// TIA Portal V18 export
// export: Created 2025-12-01T12:38:33.4037087Z, ExportSetting None, DisplayName Totally Integrated Automation Portal, DisplayVersion V18 Update 5, DisplayName TIA Portal Openness, DisplayVersion V18 Update 5, DisplayName TIA Portal Teamcenter Gateway, DisplayVersion V18, DisplayName TIA Portal Version Control Interface, DisplayVersion V18, DisplayName STEP 7 Professional, DisplayVersion V18 Update 5, DisplayName STEP 7 Safety, DisplayVersion V18, DisplayName WinCC Professional, DisplayVersion V18 Update 5
FUNCTION "ST10Cyl_interface11-20" : Void   // FC1021, LAD
{ S7_Optimized_Access := 'FALSE' }
// stored: AutoNumber false, SetENOAutomatically false
   VAR_INPUT
      AlwaysON : Bool;
      E_stop : Bool;
   END_VAR
   VAR_TEMP
      tTest : Bool;
   END_VAR
BEGIN

REGION Network 1 (SCL): Cylinder 11-20 IO Interface (SCL)

   //Cylinder11 IO   E-NG-01NGLocationCylinder
   //Input
   "ST10Cylinder".Cy[11].In.WorkPositionSensor := "iE-NG-01NGLocationCylinderInWP";
   "ST10Cylinder".Cy[11].In.HomePositionSensor := "iE-NG-01NGLocationCylinderInHP";
   //Output
   "oE-NG-01NGLocationCylinderToWP" := "ST10Cylinder".Cy[11].Out.GoWorkPosition;
   "oE-NG-01NGLocationCylinderToHP" := "ST10Cylinder".Cy[11].Out.GoHomePosition;

   //Cylinder12 IO  E-NG-02NGLocationCylinder
   //Input
   "ST10Cylinder".Cy[12].In.WorkPositionSensor := "iE-NG-02NGLocationCylinderInWP";
   "ST10Cylinder".Cy[12].In.HomePositionSensor := "iE-NG-02NGLocationCylinderInHP";
   //Output
   "oE-NG-02NGLocationCylinderToWP" := "ST10Cylinder".Cy[12].Out.GoWorkPosition;
   "oE-NG-02NGLocationCylinderToHP" := "ST10Cylinder".Cy[12].Out.GoHomePosition;

   //Cylinder13 IO  F-ROOBT1Gripper1Cylinder
   //Input
   "KukaRobot1_CtrlDB".sPLCtoROB.User.Gripper.DI129_Grip1WP:="ST10Cylinder".Cy[13].In.WorkPositionSensor := "iF-ROOBT1Gripper1CylinderInWP" ;
   "KukaRobot1_CtrlDB".sPLCtoROB.User.Gripper.DI130_Grip1HP := "ST10Cylinder".Cy[13].In.HomePositionSensor := "iF-ROOBT1Gripper1CylinderInHP" ;//"TON".TON[0].Q;

   IF  NOT "Robot_DB".Control.Robot1GripControl THEN
       //Output
       "oF-ROOBT1Gripper1CylinderToWP" := "KukaRobot1_CtrlDB".sROBtoPLC.User.Gripper.DO129_Grip1GoWork;
       "oF-ROOBT1Gripper1CylinderToHP" := "KukaRobot1_CtrlDB".sROBtoPLC.User.Gripper.DO130_Grip1GoHome;
   ELSE
       //Output
       "oF-ROOBT1Gripper1CylinderToWP" := "ST10Cylinder".Cy[13].Out.GoWorkPosition;
       "oF-ROOBT1Gripper1CylinderToHP" := "ST10Cylinder".Cy[13].Out.GoHomePosition;
   END_IF;
   "TON".TON[0](IN:="oF-ROOBT1Gripper1CylinderToHP" AND NOT"iF-ROOBT1Gripper1CylinderInWP",PT:=T#500MS);


   //Cylinder14 IO  F-ROOBT1Gripper2Cylinder
   //Input
   "KukaRobot1_CtrlDB".sPLCtoROB.User.Gripper.DI131_Grip2WP:="ST10Cylinder".Cy[14].In.WorkPositionSensor := "iF-ROOBT1Gripper2CylinderInWP";
   "KukaRobot1_CtrlDB".sPLCtoROB.User.Gripper.DI132_Grip2HP:="ST10Cylinder".Cy[14].In.HomePositionSensor := "iF-ROOBT1Gripper2CylinderInHP";

   IF NOT "Robot_DB".Control.Robot1GripControl THEN
       //Output
       "oF-ROOBT1Gripper2CylinderToWP" :="ST10Cylinder".Cy[14].Inout.AutoGoWork:="KukaRobot1_CtrlDB".sROBtoPLC.User.Gripper.DO131_Grip2GoWork;
       "oF-ROOBT1Gripper2CylinderToHP" :="ST10Cylinder".Cy[14].Inout.AutoGoHome:="KukaRobot1_CtrlDB".sROBtoPLC.User.Gripper.DO132_Grip2GoHome;
   ELSE
       //Output
       "oF-ROOBT1Gripper2CylinderToWP" := "ST10Cylinder".Cy[14].Out.GoWorkPosition;
       "oF-ROOBT1Gripper2CylinderToHP" := "ST10Cylinder".Cy[14].Out.GoHomePosition;
   END_IF;


   //Cylinder15 IO  F-ROOBT2Gripper1Cylinder
   //Input
   "KukaRobot2_CtrlDB".sPLCtoROB.User.Gripper.DI129_Grip1WP:="ST10Cylinder".Cy[15].In.WorkPositionSensor := "iF-ROOBT2Gripper1CylinderInWP";
   "KukaRobot2_CtrlDB".sPLCtoROB.User.Gripper.DI130_Grip1HP := "ST10Cylinder".Cy[15].In.HomePositionSensor :="iF-ROOBT2Gripper1CylinderInHP";

   IF NOT "Robot_DB".Control.Robot2GripControl THEN
       //Output
       "oF-ROOBT2Gripper1CylinderToWP" :="ST10Cylinder".Cy[15].Inout.AutoGoWork:="KukaRobot2_CtrlDB".sROBtoPLC.User.Gripper.DO129_Grip1GoWork;
       "oF-ROOBT2Gripper1CylinderToHP" :="ST10Cylinder".Cy[15].Inout.AutoGoHome:="KukaRobot2_CtrlDB".sROBtoPLC.User.Gripper.DO130_Grip1GoHome;
   ELSE
       //Output
       "oF-ROOBT2Gripper1CylinderToWP" := "ST10Cylinder".Cy[15].Out.GoWorkPosition;
       "oF-ROOBT2Gripper1CylinderToHP" := "ST10Cylinder".Cy[15].Out.GoHomePosition;
   END_IF;



   //Cylinder16 IO  F-ROOBT2Gripper2Cylinder
   //Input
   "KukaRobot2_CtrlDB".sPLCtoROB.User.Gripper.DI131_Grip2WP:="ST10Cylinder".Cy[16].In.WorkPositionSensor := "iF-ROOBT2Gripper2CylinderInWP";
   "KukaRobot2_CtrlDB".sPLCtoROB.User.Gripper.DI132_Grip2HP:="ST10Cylinder".Cy[16].In.HomePositionSensor := "iF-ROOBT2Gripper2CylinderInHP";

   IF NOT "Robot_DB".Control.Robot2GripControl THEN
       //Output
       "oF-ROOBT2Gripper2CylinderToWP" :="ST10Cylinder".Cy[16].Inout.AutoGoWork:= "KukaRobot2_CtrlDB".sROBtoPLC.User.Gripper.DO131_Grip2GoWork;
       "oF-ROOBT2Gripper2CylinderToHP" :="ST10Cylinder".Cy[16].Inout.AutoGoHome:= "KukaRobot2_CtrlDB".sROBtoPLC.User.Gripper.DO132_Grip2GoHome;
   ELSE
       //Output
       "oF-ROOBT2Gripper2CylinderToWP" := "ST10Cylinder".Cy[16].Out.GoWorkPosition;
       "oF-ROOBT2Gripper2CylinderToHP" := "ST10Cylinder".Cy[16].Out.GoHomePosition;
   END_IF;

   //Cylinder17 IO  F-ROOBT3Gripper1Cylinder
   //Input
   "KukaRobot3_CtrlDB".sPLCtoROB.User.Gripper.DI129_Grip1WP:="ST10Cylinder".Cy[17].In.WorkPositionSensor := "iF-ROOBT3Gripper1CylinderInWP";
   "KukaRobot3_CtrlDB".sPLCtoROB.User.Gripper.DI130_Grip1HP:="ST10Cylinder".Cy[17].In.HomePositionSensor := "iF-ROOBT3Gripper1CylinderInHP";

   IF NOT "Robot_DB".Control.Robot3GripControl THEN
       //Output
       "oF-ROOBT3Gripper1CylinderToWP" :="ST10Cylinder".Cy[17].Inout.AutoGoWork:="KukaRobot3_CtrlDB".sROBtoPLC.User.Gripper.DO129_Grip1GoWork;
       "oF-ROOBT3Gripper1CylinderToHP" :="ST10Cylinder".Cy[17].Inout.AutoGoHome:="KukaRobot3_CtrlDB".sROBtoPLC.User.Gripper.DO130_Grip1GoHome;
   ELSE
       //Output
       "oF-ROOBT3Gripper1CylinderToWP" := "ST10Cylinder".Cy[17].Out.GoWorkPosition;
       "oF-ROOBT3Gripper1CylinderToHP" := "ST10Cylinder".Cy[17].Out.GoHomePosition;
   END_IF;


   //Cylinder18 IO  F-ROOBT3Gripper2Cylinder
   //Input
   "KukaRobot3_CtrlDB".sPLCtoROB.User.Gripper.DI131_Grip2WP:="ST10Cylinder".Cy[18].In.WorkPositionSensor := "iF-ROOBT3Gripper2CylinderInWP";
   "KukaRobot3_CtrlDB".sPLCtoROB.User.Gripper.DI132_Grip2HP := "ST10Cylinder".Cy[18].In.HomePositionSensor := "iF-ROOBT3Gripper2CylinderInHP";//"TON".TON[1].Q;

   IF NOT "Robot_DB".Control.Robot3GripControl THEN
       //Output
       "oF-ROOBT3Gripper2CylinderToWP" :="ST10Cylinder".Cy[18].Inout.AutoGoWork:="KukaRobot3_CtrlDB".sROBtoPLC.User.Gripper.DO131_Grip2GoWork;
       "oF-ROOBT3Gripper2CylinderToHP" :="ST10Cylinder".Cy[18].Inout.AutoGoHome:="KukaRobot3_CtrlDB".sROBtoPLC.User.Gripper.DO132_Grip2GoHome;
   ELSE
       //Output
       "oF-ROOBT3Gripper2CylinderToWP" := "ST10Cylinder".Cy[18].Out.GoWorkPosition;
       "oF-ROOBT3Gripper2CylinderToHP" := "ST10Cylinder".Cy[18].Out.GoHomePosition;
   END_IF;

   "TON".TON[1](IN := "oF-ROOBT3Gripper2CylinderToHP" AND NOT "iF-ROOBT3Gripper2CylinderInWP",
                PT := T#500MS);

   (*
   //Cylinder19 IO  D-washer Loading Horizontal
   //Input
   "ST10Cylinder".Cy[19].In.WorkPositionSensor := ("D-washer Loading Cylinder Middle Cylinder InHP" AND "D-washer Loading Horizontal Cylinder InWP")
                                               OR ("D-washer Loading Cylinder Middle Cylinder InWP" AND "D-washer Loading Horizontal Cylinder InWP1");
   "ST10Cylinder".Cy[19].In.HomePositionSensor := "D-washer Loading Horizontal Cylinder InHP";
   //Output
   "D-washer Loading Horizontal Cylinder ToWP" := "ST10Cylinder".Cy[19].Out.GoWorkPosition;
   "D-washer Loading Horizontal Cylinder ToHP" := "ST10Cylinder".Cy[19].Out.GoHomePosition;

   //Cylinder20 IO  D-washer Loading Cylinder Middle
   //Input
   "ST10Cylinder".Cy[20].In.WorkPositionSensor := "D-washer Loading Cylinder Middle Cylinder InWP";
   "ST10Cylinder".Cy[20].In.HomePositionSensor := "D-washer Loading Cylinder Middle Cylinder InHP";
   //Output
   "D-washer Loading Cylinder Middle Cylinder ToWP" := "ST10Cylinder".Cy[20].Out.GoWorkPosition;
   "D-washer Loading Cylinder Middle Cylinder ToHP" := "ST10Cylinder".Cy[20].Out.GoHomePosition;
   *)
END_REGION

REGION Network 2: CY11 interface E-NG-01NGLocationCylinder
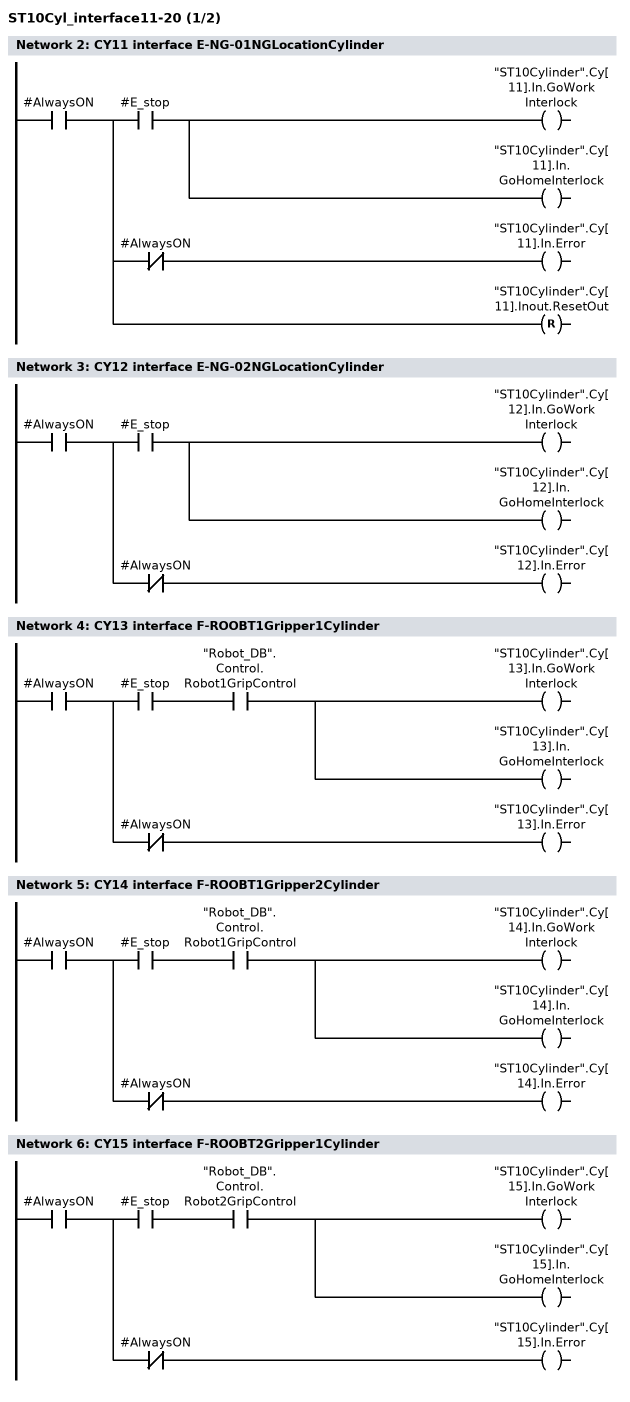
   RUNG wire#powerrail
      Contact( #AlwaysON )
      wire#w1
      Contact( #E_stop )
      wire#w2
      Coil( "ST10Cylinder".Cy[11].In.GoWorkInterlock )
   END_RUNG
   RUNG wire#w2
      Coil( "ST10Cylinder".Cy[11].In.GoHomeInterlock )
   END_RUNG
   RUNG wire#w1
      I_Contact( #AlwaysON )
      Coil( "ST10Cylinder".Cy[11].In.Error )
   END_RUNG
   RUNG wire#w1
      R_Coil( "ST10Cylinder".Cy[11].Inout.ResetOut )
   END_RUNG
   // the same network as SCL:
   "ST10Cylinder".Cy[11].In.GoWorkInterlock := #AlwaysON AND #E_stop;
   "ST10Cylinder".Cy[11].In.GoHomeInterlock := #AlwaysON AND #E_stop;
   "ST10Cylinder".Cy[11].In.Error := #AlwaysON AND NOT #AlwaysON;
   IF #AlwaysON THEN "ST10Cylinder".Cy[11].Inout.ResetOut := FALSE; END_IF;
END_REGION

REGION Network 3: CY12 interface E-NG-02NGLocationCylinder
   RUNG wire#powerrail
      Contact( #AlwaysON )
      wire#w1
      Contact( #E_stop )
      wire#w2
      Coil( "ST10Cylinder".Cy[12].In.GoWorkInterlock )
   END_RUNG
   RUNG wire#w2
      Coil( "ST10Cylinder".Cy[12].In.GoHomeInterlock )
   END_RUNG
   RUNG wire#w1
      I_Contact( #AlwaysON )
      Coil( "ST10Cylinder".Cy[12].In.Error )
   END_RUNG
   // the same network as SCL:
   "ST10Cylinder".Cy[12].In.GoWorkInterlock := #AlwaysON AND #E_stop;
   "ST10Cylinder".Cy[12].In.GoHomeInterlock := #AlwaysON AND #E_stop;
   "ST10Cylinder".Cy[12].In.Error := #AlwaysON AND NOT #AlwaysON;
END_REGION

REGION Network 4: CY13 interface F-ROOBT1Gripper1Cylinder
   RUNG wire#powerrail
      Contact( #AlwaysON )
      wire#w1
      Contact( #E_stop )
      Contact( "Robot_DB".Control.Robot1GripControl )
      wire#w2
      Coil( "ST10Cylinder".Cy[13].In.GoWorkInterlock )
   END_RUNG
   RUNG wire#w2
      Coil( "ST10Cylinder".Cy[13].In.GoHomeInterlock )
   END_RUNG
   RUNG wire#w1
      I_Contact( #AlwaysON )
      Coil( "ST10Cylinder".Cy[13].In.Error )
   END_RUNG
   // the same network as SCL:
   "ST10Cylinder".Cy[13].In.GoWorkInterlock := #AlwaysON AND #E_stop AND "Robot_DB".Control.Robot1GripControl;
   "ST10Cylinder".Cy[13].In.GoHomeInterlock := #AlwaysON AND #E_stop AND "Robot_DB".Control.Robot1GripControl;
   "ST10Cylinder".Cy[13].In.Error := #AlwaysON AND NOT #AlwaysON;
END_REGION

REGION Network 5: CY14 interface F-ROOBT1Gripper2Cylinder
   RUNG wire#powerrail
      Contact( #AlwaysON )
      wire#w1
      Contact( #E_stop )
      Contact( "Robot_DB".Control.Robot1GripControl )
      wire#w2
      Coil( "ST10Cylinder".Cy[14].In.GoWorkInterlock )
   END_RUNG
   RUNG wire#w2
      Coil( "ST10Cylinder".Cy[14].In.GoHomeInterlock )
   END_RUNG
   RUNG wire#w1
      I_Contact( #AlwaysON )
      Coil( "ST10Cylinder".Cy[14].In.Error )
   END_RUNG
   // the same network as SCL:
   "ST10Cylinder".Cy[14].In.GoWorkInterlock := #AlwaysON AND #E_stop AND "Robot_DB".Control.Robot1GripControl;
   "ST10Cylinder".Cy[14].In.GoHomeInterlock := #AlwaysON AND #E_stop AND "Robot_DB".Control.Robot1GripControl;
   "ST10Cylinder".Cy[14].In.Error := #AlwaysON AND NOT #AlwaysON;
END_REGION

REGION Network 6: CY15 interface F-ROOBT2Gripper1Cylinder
   RUNG wire#powerrail
      Contact( #AlwaysON )
      wire#w1
      Contact( #E_stop )
      Contact( "Robot_DB".Control.Robot2GripControl )
      wire#w2
      Coil( "ST10Cylinder".Cy[15].In.GoWorkInterlock )
   END_RUNG
   RUNG wire#w2
      Coil( "ST10Cylinder".Cy[15].In.GoHomeInterlock )
   END_RUNG
   RUNG wire#w1
      I_Contact( #AlwaysON )
      Coil( "ST10Cylinder".Cy[15].In.Error )
   END_RUNG
   // the same network as SCL:
   "ST10Cylinder".Cy[15].In.GoWorkInterlock := #AlwaysON AND #E_stop AND "Robot_DB".Control.Robot2GripControl;
   "ST10Cylinder".Cy[15].In.GoHomeInterlock := #AlwaysON AND #E_stop AND "Robot_DB".Control.Robot2GripControl;
   "ST10Cylinder".Cy[15].In.Error := #AlwaysON AND NOT #AlwaysON;
END_REGION

REGION Network 7: CY16 interface F-ROOBT2Gripper2Cylinder
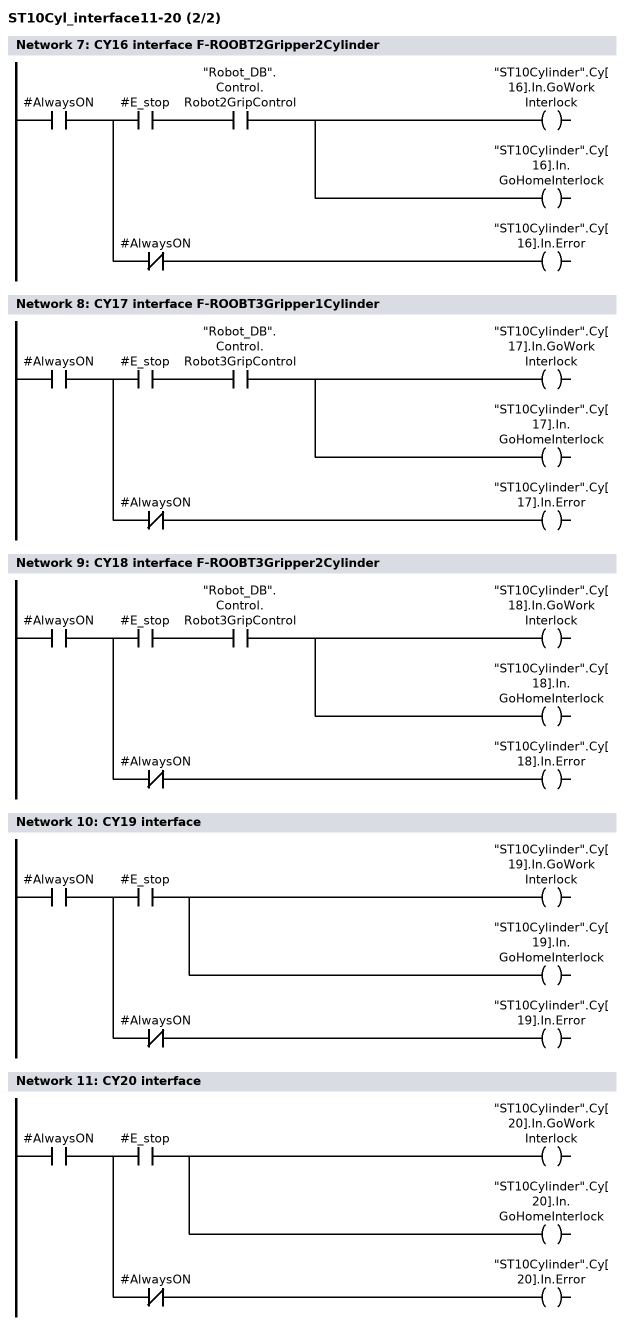
   RUNG wire#powerrail
      Contact( #AlwaysON )
      wire#w1
      Contact( #E_stop )
      Contact( "Robot_DB".Control.Robot2GripControl )
      wire#w2
      Coil( "ST10Cylinder".Cy[16].In.GoWorkInterlock )
   END_RUNG
   RUNG wire#w2
      Coil( "ST10Cylinder".Cy[16].In.GoHomeInterlock )
   END_RUNG
   RUNG wire#w1
      I_Contact( #AlwaysON )
      Coil( "ST10Cylinder".Cy[16].In.Error )
   END_RUNG
   // the same network as SCL:
   "ST10Cylinder".Cy[16].In.GoWorkInterlock := #AlwaysON AND #E_stop AND "Robot_DB".Control.Robot2GripControl;
   "ST10Cylinder".Cy[16].In.GoHomeInterlock := #AlwaysON AND #E_stop AND "Robot_DB".Control.Robot2GripControl;
   "ST10Cylinder".Cy[16].In.Error := #AlwaysON AND NOT #AlwaysON;
END_REGION

REGION Network 8: CY17 interface F-ROOBT3Gripper1Cylinder
   RUNG wire#powerrail
      Contact( #AlwaysON )
      wire#w1
      Contact( #E_stop )
      Contact( "Robot_DB".Control.Robot3GripControl )
      wire#w2
      Coil( "ST10Cylinder".Cy[17].In.GoWorkInterlock )
   END_RUNG
   RUNG wire#w2
      Coil( "ST10Cylinder".Cy[17].In.GoHomeInterlock )
   END_RUNG
   RUNG wire#w1
      I_Contact( #AlwaysON )
      Coil( "ST10Cylinder".Cy[17].In.Error )
   END_RUNG
   // the same network as SCL:
   "ST10Cylinder".Cy[17].In.GoWorkInterlock := #AlwaysON AND #E_stop AND "Robot_DB".Control.Robot3GripControl;
   "ST10Cylinder".Cy[17].In.GoHomeInterlock := #AlwaysON AND #E_stop AND "Robot_DB".Control.Robot3GripControl;
   "ST10Cylinder".Cy[17].In.Error := #AlwaysON AND NOT #AlwaysON;
END_REGION

REGION Network 9: CY18 interface F-ROOBT3Gripper2Cylinder
   RUNG wire#powerrail
      Contact( #AlwaysON )
      wire#w1
      Contact( #E_stop )
      Contact( "Robot_DB".Control.Robot3GripControl )
      wire#w2
      Coil( "ST10Cylinder".Cy[18].In.GoWorkInterlock )
   END_RUNG
   RUNG wire#w2
      Coil( "ST10Cylinder".Cy[18].In.GoHomeInterlock )
   END_RUNG
   RUNG wire#w1
      I_Contact( #AlwaysON )
      Coil( "ST10Cylinder".Cy[18].In.Error )
   END_RUNG
   // the same network as SCL:
   "ST10Cylinder".Cy[18].In.GoWorkInterlock := #AlwaysON AND #E_stop AND "Robot_DB".Control.Robot3GripControl;
   "ST10Cylinder".Cy[18].In.GoHomeInterlock := #AlwaysON AND #E_stop AND "Robot_DB".Control.Robot3GripControl;
   "ST10Cylinder".Cy[18].In.Error := #AlwaysON AND NOT #AlwaysON;
END_REGION

REGION Network 10: CY19 interface
   RUNG wire#powerrail
      Contact( #AlwaysON )
      wire#w1
      Contact( #E_stop )
      wire#w2
      Coil( "ST10Cylinder".Cy[19].In.GoWorkInterlock )
   END_RUNG
   RUNG wire#w2
      Coil( "ST10Cylinder".Cy[19].In.GoHomeInterlock )
   END_RUNG
   RUNG wire#w1
      I_Contact( #AlwaysON )
      Coil( "ST10Cylinder".Cy[19].In.Error )
   END_RUNG
   // the same network as SCL:
   "ST10Cylinder".Cy[19].In.GoWorkInterlock := #AlwaysON AND #E_stop;
   "ST10Cylinder".Cy[19].In.GoHomeInterlock := #AlwaysON AND #E_stop;
   "ST10Cylinder".Cy[19].In.Error := #AlwaysON AND NOT #AlwaysON;
END_REGION

REGION Network 11: CY20 interface
   RUNG wire#powerrail
      Contact( #AlwaysON )
      wire#w1
      Contact( #E_stop )
      wire#w2
      Coil( "ST10Cylinder".Cy[20].In.GoWorkInterlock )
   END_RUNG
   RUNG wire#w2
      Coil( "ST10Cylinder".Cy[20].In.GoHomeInterlock )
   END_RUNG
   RUNG wire#w1
      I_Contact( #AlwaysON )
      Coil( "ST10Cylinder".Cy[20].In.Error )
   END_RUNG
   // the same network as SCL:
   "ST10Cylinder".Cy[20].In.GoWorkInterlock := #AlwaysON AND #E_stop;
   "ST10Cylinder".Cy[20].In.GoHomeInterlock := #AlwaysON AND #E_stop;
   "ST10Cylinder".Cy[20].In.Error := #AlwaysON AND NOT #AlwaysON;
END_REGION
END_FUNCTION
